// TwinCAT 3 PLC project Untitled1
// ProgramVersion: 3.1.4024.0
// libraries:
//   Tc2_MC2, * (Beckhoff Automation GmbH)
//   Tc2_Standard, * (Beckhoff Automation GmbH)
//   Tc2_System, * (Beckhoff Automation GmbH)
//   Tc3_Module, * (Beckhoff Automation GmbH)
// project tree:
//   GVLs/ GVL.TcGVL
//   / PlcTask.TcTTO
//   POUs/ FB_AxisBase.TcPOU, FB_MoveVelocity.TcPOU, MAIN.TcPOU
// real-time tasks:
//   TASK PlcTask: cycle T#10ms, priority 20, ADS port 350
// motion (NC):
//   TASK NC-Task 1 SAF: cycle T#2ms, priority 4, ADS port 501
//   TASK NC-Task 1 SVB: cycle T#10ms, priority 8, ADS port 511
//   AXIS Achse 1 (id 1)
//     OtherSettings: AllowMotionCmdToSlave=true
//     encoder EncType=1
//     drive DrvType=5
//       Analog: TorqueSetpointScale=10, ScaleFactorActTorque=0.1
//       TimeComp: TaskDelayCycles=1
//     controller CtrType=1
//       CtrPara: PriorControlFactor=1
//         Observer: BandWidth=20
// variable links:
//   Untitled1/Untitled1 Instance <-> NC-Task 1 SAF/Axes/Achse 1
//     PlcTask Inputs/GVL.axis_a.NcToPlc <-> Outputs/ToPlc
//     PlcTask Outputs/GVL.axis_a.PlcToNc <-> Inputs/FromPlc

CONFIGURATION Untitled1
    RESOURCE PLC ON TwinCAT3
        TASK PlcTask(INTERVAL := T#10ms, PRIORITY := 20);
        PROGRAM MAIN WITH PlcTask : MAIN;
    END_RESOURCE
END_CONFIGURATION

// ---- GVLs/GVL.TcGVL
{attribute 'qualified_only'}
VAR_GLOBAL
	axis_a : AXIS_REF;
END_VAR

// ---- POUs/MAIN.TcPOU
PROGRAM MAIN
VAR
	fb_velocity : FB_MoveVelocity;
	//fb_test : FB_AxisBase;
END_VAR

fb_velocity(axis_ref := GVL.axis_a);
//fb_test(axis_ref := GVL.axis_a);

END_PROGRAM

// ---- POUs/FB_MoveVelocity.TcPOU
FUNCTION_BLOCK FB_MoveVelocity EXTENDS FB_AxisBase
VAR_INPUT
	bStartVelo		: BOOL;
	fVelocity		: LREAL := 100; // mm/s
END_VAR
VAR_OUTPUT
END_VAR
VAR_IN_OUT
	axis_ref : AXIS_REF;
END_VAR
VAR
	m_fb_velo	: MC_MoveVelocity;
END_VAR

SUPER^(_axis_ref := axis_ref);

m_fb_velo(
	Axis := axis_ref,
	Execute := bStartVelo,
	Velocity := fVelocity
	);
	
bStartVelo := FALSE;

END_FUNCTION_BLOCK

// ---- POUs/FB_AxisBase.TcPOU
FUNCTION_BLOCK FB_AxisBase
VAR_INPUT
	_axis_ref : REFERENCE TO AXIS_REF;
	bPowerEnable 	: BOOL := TRUE;
	bStop			: BOOL;
	bReset 			: BOOL;
	fPowerOverride	: LREAL := 100;
END_VAR
VAR_OUTPUT
END_VAR
//VAR_IN_OUT
//	axis_ref : AXIS_REF;
//END_VAR
VAR
	m_fb_power 	: MC_Power;
	m_fb_reset	: MC_Reset;
	m_fb_stop  	: MC_Stop;
	
	

	m_axis_status : ST_AxisStatus;
	m_state : ST_McOutputs;
	
	st_fbMcStopOut: ST_McOutputs;
	
END_VAR

_axis_ref.ReadStatus();
m_axis_status := _axis_ref.Status;

// Reglerfreigabe
m_fb_power(
	Axis := _axis_ref,
	Enable := bPowerEnable,
	Override := fPowerOverride,
	Enable_Positive := TRUE,
	Enable_Negative := TRUE,
	);
	
m_fb_reset(
	Axis := _axis_ref,
	Execute := bReset
	);

	
m_fb_stop(
	Axis := _axis_ref,
	Execute := bStop,
	);


bStop := FALSE;
bReset := FALSE;

END_FUNCTION_BLOCK
